TYPE ST_PowerStack_Events :
STRUCT
	//INFO
	b_CoolingDerating				: BOOL;
	b_PlimitShiftingActive			: BOOL;
	
	//Warnings
	b_DCdeviationHigh				: BOOL;
	b_TemperatureWarning			: BOOL;
	b_OvercurrentWarning			: BOOL;
	b_UndervoltageWarning			: BOOL;
	b_OvervoltageWarning			: BOOL;
	b_TemperatureDeviationHigh		: BOOL;
	b_PlimitShutdownWarning			: BOOL;
	
	b_MasterWarning					: BOOL;
	b_SlaveWarning					: BOOL;
	b_GridCodeWarning				: BOOL;
	
	//faults
	b_UnderFreqFault				: BOOL;
	b_OverFreqFault					: BOOL;
	b_UnderVoltageFault				: BOOL;
	b_OverVoltageFault				: BOOL;
	b_OvercurrentFault				: BOOL;
	b_PlimitShutdown				: BOOL;
	b_TemperatureFault				: BOOL;
	b_MasterFault					: BOOL;
	b_SlaveFault					: BOOL;
	b_NetcontactorFault				: BOOL;
	
	
	b_startupTimeOut				: BOOL;
	b_ShutdownTimeOut				: BOOL;
	
	ui_shutdownRemainingTime		: UINT;
END_STRUCT
END_TYPE

(* stored: Version 1.1.0.1, ProductVersion 3.1.4026.18
   DUT ST_PowerStack_Events: Id {994a41d6-c4af-4702-8fba-3713ad71e194} *)
